// TIA Portal V18 export
TYPE "PLCtoMES_PrintExchange_ext"
// stored: IsFailsafeCompliant false
   STRUCT
      Load_PrintReq : Bool;   // 请求下发打标数据
      Load_DataMatrixCheckReq : Bool;   // 二维码内容与主零件码比对请求
      Load_Spare : Bool;   // Spare
      Load_Spare_1 : Bool;   // Spare
      Load_Spare_2 : Bool;   // Spare
      Load_Spare_3 : Bool;   // Spare
      Load_Spare_4 : Bool;   // Spare
      Load_Spare_5 : Bool;   // Spare
      Spare : Byte;   // Spare
   END_STRUCT;
END_TYPE
